(*------------- Simple TCP/IP client application. Adapt this code to match your needs. -----*)
FUNCTION_BLOCK FB_ClientApplication
VAR_IN_OUT
	fbTx 		: FB_FrameFifo;(* TX fifo *)
	fbRx 		: FB_FrameFifo;(* RX fifo *)
	fbLog		: FB_LogFifo;(* Log message fifo *)
END_VAR
VAR
	sToServer	: T_MaxString := '';
	sFromServer	: T_MaxString := '';
	sLogMessage	: T_MaxString := '';
	nCounter	: UDINT;
	fbSndTimer	: TON;
END_VAR

(*------------------- Send cyclic message strings ------------------------------------*)
fbSndTimer( IN := TRUE, PT := PLCPRJ_SEND_CYCLE_TIME );
IF fbSndTimer.Q THEN(* Send string to server *)
	fbSndTimer( IN := FALSE );

	nCounter := nCounter  + 1;
	sToServer := 'PL.FB$0D$0A';
 
	fbTx.AddTail( sPut := sToServer );(* Put string to the tx fifo *)
	IF NOT fbTx.bOk THEN(* TX fifo overflow => log error *)
		fbLog.Error( sMessage := 'FB_FrameFifo(sender)', nErrID := PLCPRJ_ERROR_SENDFIFO_OVERFLOW );
	END_IF

END_IF

(*--------------------- Get received message strings --------------------------------*)
REPEAT
	fbRx.RemoveHead( );(* Fetch string from rx fifo *)
	IF fbRx.bOk THEN(* Success *)

		(* TODO: Implement receive data handler *)
		sFromServer := fbRx.sGet; 		
		
	END_IF
UNTIL NOT fbRx.bOk
END_REPEAT

(*------------------------------- Get log/error messages from log fifo -------------*)
REPEAT
	fbLog.Remove( );
	IF fbLog.bOk THEN
		
		(* TODO: Implement log message handler *)
		sLogMessage := fbLog.sGet; 
		
	END_IF
UNTIL NOT fbLog.bOk
END_REPEAT

END_FUNCTION_BLOCK

(* stored: Version 1.1.0.1
   POU FB_ClientApplication: Id {e1f59b55-4ed3-4201-89c5-639c8eca1b2b}, SpecialFunc None *)
